PROGRAM MAIN
VAR
	App : TeamsApp;
END_VAR

App.Run();

END_PROGRAM

(* stored: Version 1.1.0.1, ProductVersion 3.1.4024.9
   POU MAIN: Id {f430142b-5594-40e1-be88-c972d031e187}, SpecialFunc None *)
